PROGRAM MAIN
VAR
	fbRamp1: FB_Ramp;
	fbRamp2: FB_Ramp;
	fbShiftArray: FB_ShiftArray;
	fbRunningLight: FB_RunningLight;
	Ramp1 : INT;
	Ramp2 : INT;
	RunningLight1: BOOL;
	RunningLight2: BOOL;
	RunningLight3: BOOL;
	RunningLight4: BOOL;
	RunningLight5: BOOL;
	
END_VAR

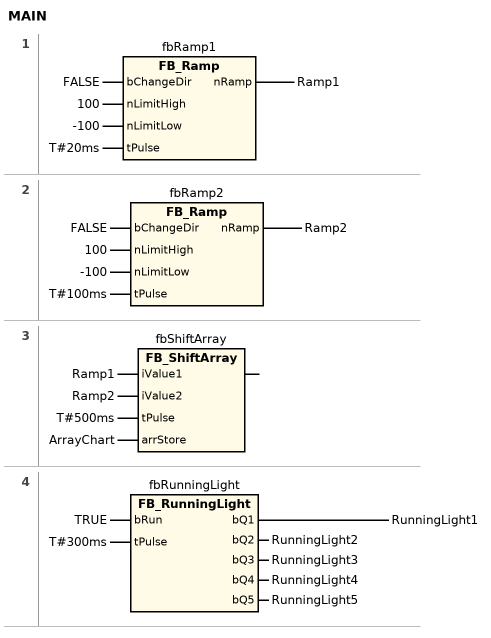
// NETWORK 1
fbRamp1(bChangeDir := FALSE, nLimitHigh := 100, nLimitLow := -100, tPulse := T#20ms); // FB_Ramp
Ramp1 := fbRamp1.nRamp;

// NETWORK 2
fbRamp2(bChangeDir := FALSE, nLimitHigh := 100, nLimitLow := -100, tPulse := T#100ms); // FB_Ramp
Ramp2 := fbRamp2.nRamp;

// NETWORK 3
fbShiftArray(iValue1 := Ramp1, iValue2 := Ramp2, tPulse := T#500ms, arrStore := ArrayChart); // FB_ShiftArray

// NETWORK 4
fbRunningLight(
    bRun := TRUE,
    tPulse := T#300ms,
    bQ2 => RunningLight2,
    bQ3 => RunningLight3,
    bQ4 => RunningLight4,
    bQ5 => RunningLight5); // FB_RunningLight
RunningLight1 := fbRunningLight.bQ1;

END_PROGRAM

(* stored: Version 1.1.0.1, ProductVersion 3.1.4022.7
   POU MAIN: Id {8234e2d6-d2f6-48c1-ac1e-99c81a5a71a9}, SpecialFunc None *)
